SYSTEM SystemTests
  (* Version 1.0, 2018-08-29, Alois Zoitl, Johannes Kepler University, initial API and implementation and/or initial documentation *)
  APPLICATION Timing (* Small test application for measuring the execution time of a few fbs for evaluating runtime performance *)
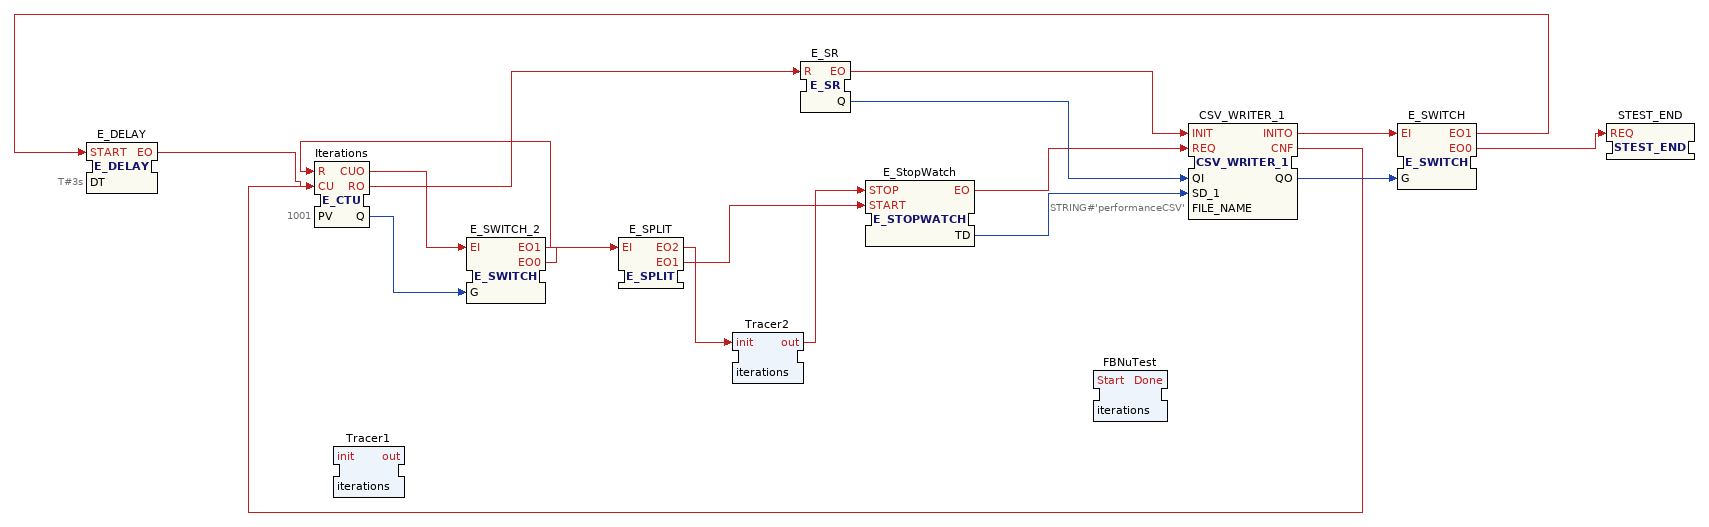
    FBS
      CSV_WRITER_1 : CSV_WRITER_1(FILE_NAME := STRING#'performanceCSV');
      E_SR : E_SR;
      E_SWITCH_2 : E_SWITCH;
      Iterations : E_CTU(PV := 1001);
      STEST_END : STEST_END;
      E_SWITCH : E_SWITCH;
      E_StopWatch : E_STOPWATCH;
      E_SPLIT : E_SPLIT;
      E_DELAY : E_DELAY(DT := T#3s);
    END_FBS
    SUBAPPLICATION FBNuTest
      EVENT_INPUT
        Start;
      END_EVENT
      EVENT_OUTPUT
        Done;
      END_EVENT
      VAR_INPUT
        iterations : UINT := UINT#100;
      END_VAR
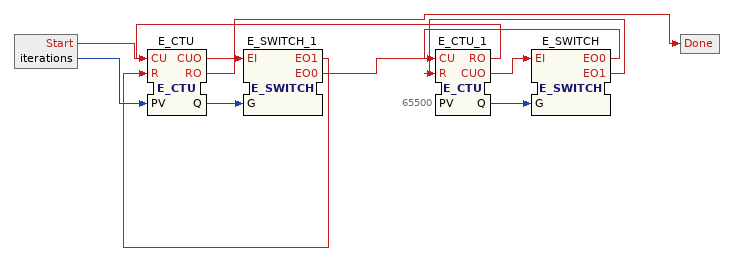
      FBS
        E_CTU : E_CTU;
        E_SWITCH_1 : E_SWITCH;
        E_SWITCH : E_SWITCH;
        E_CTU_1 : E_CTU(PV := 65500);
      END_FBS
      EVENT_CONNECTIONS
        E_CTU_1.RO TO E_CTU.CU;
        E_SWITCH_1.EO1 TO E_CTU.R;
        E_CTU.CUO TO E_SWITCH_1.EI;
        E_SWITCH_1.EO0 TO E_CTU_1.CU;
        E_CTU_1.CUO TO E_SWITCH.EI;
        E_SWITCH.EO0 TO E_CTU_1.CU;
        E_SWITCH.EO1 TO E_CTU_1.R;
        Start TO E_CTU.CU;
        E_CTU.RO TO Done;
      END_CONNECTIONS
      DATA_CONNECTIONS
        E_CTU.Q TO E_SWITCH_1.G;
        E_CTU_1.Q TO E_SWITCH.G;
        iterations TO E_CTU.PV;
      END_CONNECTIONS
    END_SUBAPPLICATION
    SUBAPPLICATION Tracer1
      EVENT_INPUT
        init;
      END_EVENT
      EVENT_OUTPUT
        out;
      END_EVENT
      VAR_INPUT
        iterations : UINT := UINT#1000;
      END_VAR
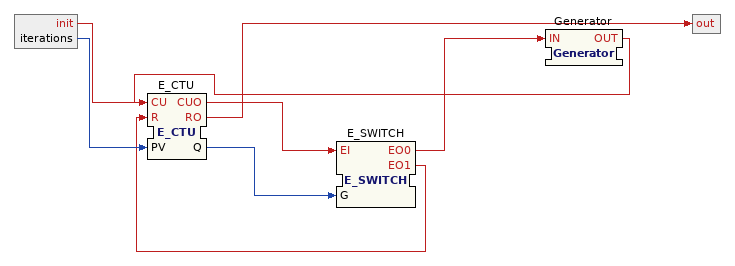
      FBS
        Generator : performance::Generator;
        E_CTU : E_CTU;
        E_SWITCH : E_SWITCH;
      END_FBS
      EVENT_CONNECTIONS
        init TO E_CTU.CU;
        E_CTU.CUO TO E_SWITCH.EI;
        E_SWITCH.EO0 TO Generator.IN;
        E_CTU.RO TO out;
        Generator.OUT TO E_CTU.CU;
        E_SWITCH.EO1 TO E_CTU.R;
      END_CONNECTIONS
      DATA_CONNECTIONS
        iterations TO E_CTU.PV;
        E_CTU.Q TO E_SWITCH.G;
      END_CONNECTIONS
    END_SUBAPPLICATION
    SUBAPPLICATION Tracer2
      EVENT_INPUT
        init;
      END_EVENT
      EVENT_OUTPUT
        out;
      END_EVENT
      VAR_INPUT
        iterations : UINT := UINT#1001;
      END_VAR
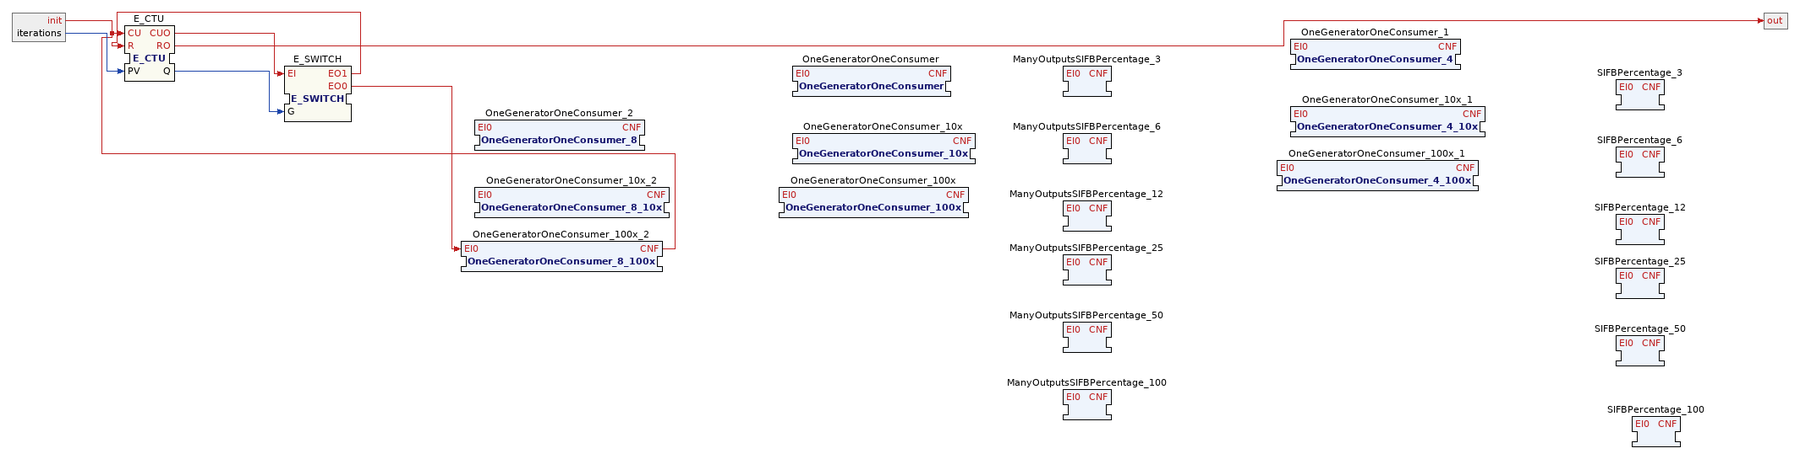
      FBS
        E_CTU : E_CTU;
        E_SWITCH : E_SWITCH;
      END_FBS
      SUBAPPS
        OneGeneratorOneConsumer : OneGeneratorOneConsumer;
        OneGeneratorOneConsumer_10x : OneGeneratorOneConsumer_10x;
        OneGeneratorOneConsumer_100x : OneGeneratorOneConsumer_100x;
        OneGeneratorOneConsumer_1 : OneGeneratorOneConsumer_4;
        OneGeneratorOneConsumer_10x_1 : OneGeneratorOneConsumer_4_10x;
        OneGeneratorOneConsumer_100x_1 : OneGeneratorOneConsumer_4_100x;
        OneGeneratorOneConsumer_100x_2 : OneGeneratorOneConsumer_8_100x;
        OneGeneratorOneConsumer_2 : OneGeneratorOneConsumer_8;
        OneGeneratorOneConsumer_10x_2 : OneGeneratorOneConsumer_8_10x;
      END_SUBAPPS
      SUBAPPLICATION SIFBPercentage_3
        {SET_ATTRIBUTE(Attribute1, )}
        EVENT_INPUT
          EI0;
        END_EVENT
        EVENT_OUTPUT
          CNF;
        END_EVENT
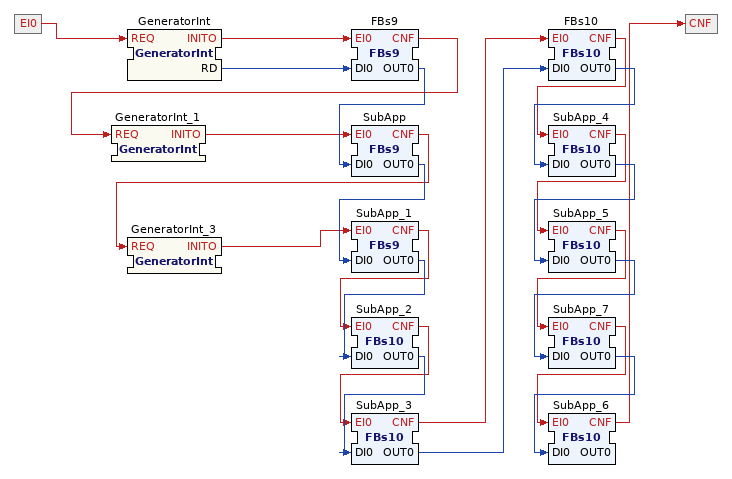
        FBS
          GeneratorInt : performance::GeneratorInt;
          GeneratorInt_1 : performance::GeneratorInt;
          GeneratorInt_3 : performance::GeneratorInt;
        END_FBS
        SUBAPPS
          FBs9 : FBs9;
          SubApp : FBs9;
          SubApp_1 : FBs9;
          SubApp_2 : FBs10;
          SubApp_3 : FBs10;
          SubApp_4 : FBs10;
          SubApp_5 : FBs10;
          SubApp_6 : FBs10;
          SubApp_7 : FBs10;
          FBs10 : FBs10;
        END_SUBAPPS
        EVENT_CONNECTIONS
          EI0 TO GeneratorInt.REQ;
          SubApp_2.CNF TO SubApp_3.EI0;
          SubApp_4.CNF TO SubApp_5.EI0;
          SubApp_5.CNF TO SubApp_7.EI0;
          SubApp_7.CNF TO SubApp_6.EI0;
          SubApp_3.CNF TO FBs10.EI0;
          FBs10.CNF TO SubApp_4.EI0;
          SubApp_6.CNF TO CNF;
          FBs9.CNF TO GeneratorInt_1.REQ;
          SubApp.CNF TO GeneratorInt_3.REQ;
          GeneratorInt_1.INITO TO SubApp.EI0;
          GeneratorInt.INITO TO FBs9.EI0;
          GeneratorInt_3.INITO TO SubApp_1.EI0;
          SubApp_1.CNF TO SubApp_2.EI0;
        END_CONNECTIONS
        DATA_CONNECTIONS
          SubApp_2.OUT0 TO SubApp_3.DI0;
          SubApp_1.OUT0 TO SubApp_2.DI0;
          SubApp.OUT0 TO SubApp_1.DI0;
          SubApp_7.OUT0 TO SubApp_6.DI0;
          SubApp_4.OUT0 TO SubApp_5.DI0;
          SubApp_5.OUT0 TO SubApp_7.DI0;
          FBs10.OUT0 TO SubApp_4.DI0;
          SubApp_3.OUT0 TO FBs10.DI0;
          GeneratorInt.RD TO FBs9.DI0;
          FBs9.OUT0 TO SubApp.DI0;
        END_CONNECTIONS
      END_SUBAPPLICATION
      SUBAPPLICATION SIFBPercentage_6
        {SET_ATTRIBUTE(Attribute1, )}
        EVENT_INPUT
          EI0;
        END_EVENT
        EVENT_OUTPUT
          CNF;
        END_EVENT
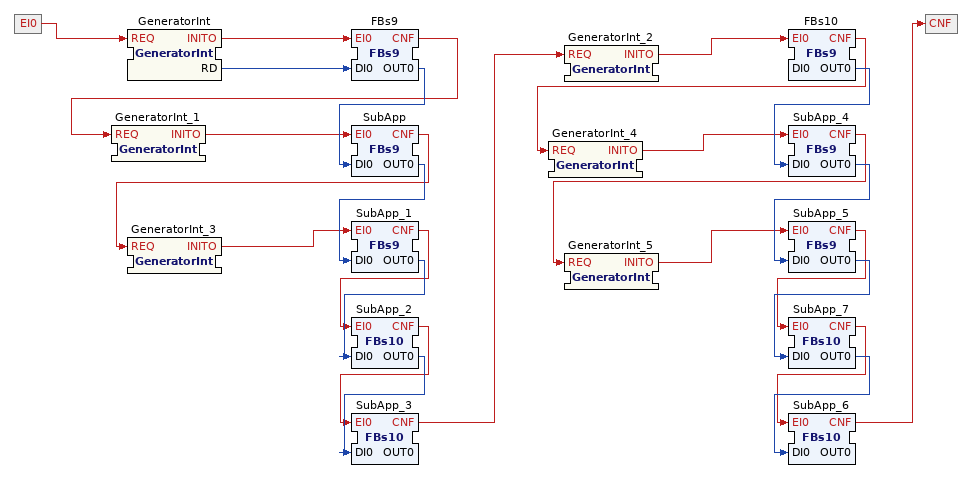
        FBS
          GeneratorInt : performance::GeneratorInt;
          GeneratorInt_1 : performance::GeneratorInt;
          GeneratorInt_3 : performance::GeneratorInt;
          GeneratorInt_2 : performance::GeneratorInt;
          GeneratorInt_4 : performance::GeneratorInt;
          GeneratorInt_5 : performance::GeneratorInt;
        END_FBS
        SUBAPPS
          FBs9 : FBs9;
          SubApp : FBs9;
          SubApp_1 : FBs9;
          SubApp_2 : FBs10;
          SubApp_3 : FBs10;
          SubApp_4 : FBs9;
          SubApp_5 : FBs9;
          SubApp_6 : FBs10;
          SubApp_7 : FBs10;
          FBs10 : FBs9;
        END_SUBAPPS
        EVENT_CONNECTIONS
          EI0 TO GeneratorInt.REQ;
          SubApp_2.CNF TO SubApp_3.EI0;
          SubApp_4.CNF TO GeneratorInt_5.REQ;
          SubApp_5.CNF TO SubApp_7.EI0;
          SubApp_7.CNF TO SubApp_6.EI0;
          FBs10.CNF TO GeneratorInt_4.REQ;
          SubApp_6.CNF TO CNF;
          FBs9.CNF TO GeneratorInt_1.REQ;
          SubApp.CNF TO GeneratorInt_3.REQ;
          GeneratorInt_1.INITO TO SubApp.EI0;
          GeneratorInt.INITO TO FBs9.EI0;
          GeneratorInt_3.INITO TO SubApp_1.EI0;
          GeneratorInt_2.INITO TO FBs10.EI0;
          GeneratorInt_4.INITO TO SubApp_4.EI0;
          GeneratorInt_5.INITO TO SubApp_5.EI0;
          SubApp_3.CNF TO GeneratorInt_2.REQ;
          SubApp_1.CNF TO SubApp_2.EI0;
        END_CONNECTIONS
        DATA_CONNECTIONS
          SubApp_2.OUT0 TO SubApp_3.DI0;
          SubApp_1.OUT0 TO SubApp_2.DI0;
          SubApp.OUT0 TO SubApp_1.DI0;
          SubApp_7.OUT0 TO SubApp_6.DI0;
          SubApp_4.OUT0 TO SubApp_5.DI0;
          SubApp_5.OUT0 TO SubApp_7.DI0;
          FBs10.OUT0 TO SubApp_4.DI0;
          GeneratorInt.RD TO FBs9.DI0;
          FBs9.OUT0 TO SubApp.DI0;
        END_CONNECTIONS
      END_SUBAPPLICATION
      SUBAPPLICATION SIFBPercentage_12
        {SET_ATTRIBUTE(Attribute1, )}
        EVENT_INPUT
          EI0;
        END_EVENT
        EVENT_OUTPUT
          CNF;
        END_EVENT
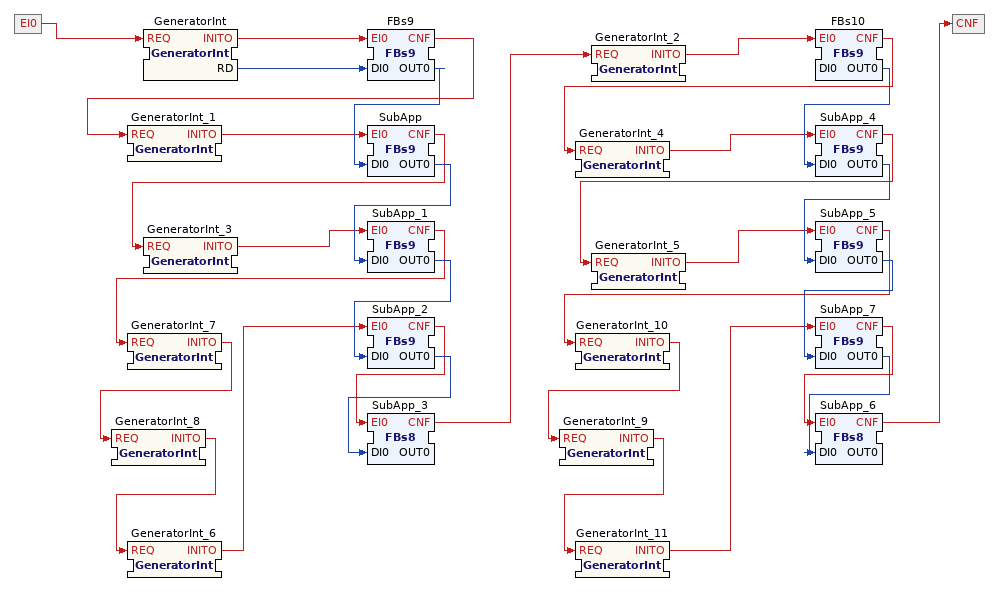
        FBS
          GeneratorInt : performance::GeneratorInt;
          GeneratorInt_1 : performance::GeneratorInt;
          GeneratorInt_3 : performance::GeneratorInt;
          GeneratorInt_2 : performance::GeneratorInt;
          GeneratorInt_4 : performance::GeneratorInt;
          GeneratorInt_5 : performance::GeneratorInt;
          GeneratorInt_6 : performance::GeneratorInt;
          GeneratorInt_7 : performance::GeneratorInt;
          GeneratorInt_8 : performance::GeneratorInt;
          GeneratorInt_9 : performance::GeneratorInt;
          GeneratorInt_10 : performance::GeneratorInt;
          GeneratorInt_11 : performance::GeneratorInt;
        END_FBS
        SUBAPPS
          FBs9 : FBs9;
          SubApp : FBs9;
          SubApp_1 : FBs9;
          SubApp_2 : FBs9;
          SubApp_3 : FBs8;
          SubApp_4 : FBs9;
          SubApp_5 : FBs9;
          SubApp_6 : FBs8;
          SubApp_7 : FBs9;
          FBs10 : FBs9;
        END_SUBAPPS
        EVENT_CONNECTIONS
          EI0 TO GeneratorInt.REQ;
          SubApp_2.CNF TO SubApp_3.EI0;
          SubApp_4.CNF TO GeneratorInt_5.REQ;
          SubApp_5.CNF TO GeneratorInt_10.REQ;
          SubApp_7.CNF TO SubApp_6.EI0;
          FBs10.CNF TO GeneratorInt_4.REQ;
          SubApp_6.CNF TO CNF;
          FBs9.CNF TO GeneratorInt_1.REQ;
          SubApp.CNF TO GeneratorInt_3.REQ;
          GeneratorInt_1.INITO TO SubApp.EI0;
          GeneratorInt.INITO TO FBs9.EI0;
          GeneratorInt_3.INITO TO SubApp_1.EI0;
          GeneratorInt_2.INITO TO FBs10.EI0;
          GeneratorInt_4.INITO TO SubApp_4.EI0;
          GeneratorInt_5.INITO TO SubApp_5.EI0;
          SubApp_3.CNF TO GeneratorInt_2.REQ;
          SubApp_1.CNF TO GeneratorInt_7.REQ;
          GeneratorInt_7.INITO TO GeneratorInt_8.REQ;
          GeneratorInt_8.INITO TO GeneratorInt_6.REQ;
          GeneratorInt_6.INITO TO SubApp_2.EI0;
          GeneratorInt_10.INITO TO GeneratorInt_9.REQ;
          GeneratorInt_9.INITO TO GeneratorInt_11.REQ;
          GeneratorInt_11.INITO TO SubApp_7.EI0;
        END_CONNECTIONS
        DATA_CONNECTIONS
          SubApp_2.OUT0 TO SubApp_3.DI0;
          SubApp_1.OUT0 TO SubApp_2.DI0;
          SubApp.OUT0 TO SubApp_1.DI0;
          SubApp_7.OUT0 TO SubApp_6.DI0;
          SubApp_4.OUT0 TO SubApp_5.DI0;
          SubApp_5.OUT0 TO SubApp_7.DI0;
          FBs10.OUT0 TO SubApp_4.DI0;
          GeneratorInt.RD TO FBs9.DI0;
          FBs9.OUT0 TO SubApp.DI0;
        END_CONNECTIONS
      END_SUBAPPLICATION
      SUBAPPLICATION SIFBPercentage_25
        {SET_ATTRIBUTE(Attribute1, )}
        EVENT_INPUT
          EI0;
        END_EVENT
        EVENT_OUTPUT
          CNF;
        END_EVENT
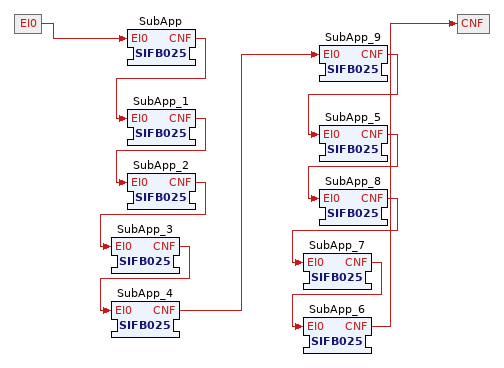
        SUBAPPS
          SubApp : SIFB025;
          SubApp_1 : SIFB025;
          SubApp_2 : SIFB025;
          SubApp_3 : SIFB025;
          SubApp_4 : SIFB025;
          SubApp_5 : SIFB025;
          SubApp_6 : SIFB025;
          SubApp_7 : SIFB025;
          SubApp_8 : SIFB025;
          SubApp_9 : SIFB025;
        END_SUBAPPS
        EVENT_CONNECTIONS
          SubApp_3.CNF TO SubApp_4.EI0;
          SubApp_2.CNF TO SubApp_3.EI0;
          SubApp_1.CNF TO SubApp_2.EI0;
          SubApp.CNF TO SubApp_1.EI0;
          SubApp_5.CNF TO SubApp_8.EI0;
          SubApp_8.CNF TO SubApp_7.EI0;
          SubApp_7.CNF TO SubApp_6.EI0;
          SubApp_9.CNF TO SubApp_5.EI0;
          SubApp_4.CNF TO SubApp_9.EI0;
          EI0 TO SubApp.EI0;
          SubApp_6.CNF TO CNF;
        END_CONNECTIONS
      END_SUBAPPLICATION
      SUBAPPLICATION SIFBPercentage_50
        {SET_ATTRIBUTE(Attribute1, )}
        EVENT_INPUT
          EI0;
        END_EVENT
        EVENT_OUTPUT
          CNF;
        END_EVENT
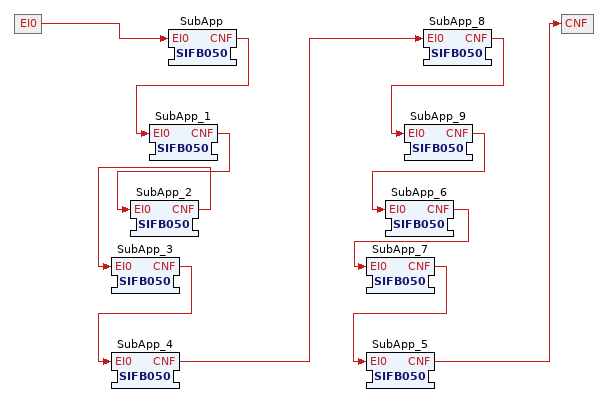
        SUBAPPS
          SubApp : SIFB050;
          SubApp_1 : SIFB050;
          SubApp_2 : SIFB050;
          SubApp_3 : SIFB050;
          SubApp_4 : SIFB050;
          SubApp_5 : SIFB050;
          SubApp_6 : SIFB050;
          SubApp_7 : SIFB050;
          SubApp_8 : SIFB050;
          SubApp_9 : SIFB050;
        END_SUBAPPS
        EVENT_CONNECTIONS
          SubApp.CNF TO SubApp_1.EI0;
          SubApp_1.CNF TO SubApp_2.EI0;
          SubApp_2.CNF TO SubApp_3.EI0;
          SubApp_3.CNF TO SubApp_4.EI0;
          SubApp_8.CNF TO SubApp_9.EI0;
          SubApp_9.CNF TO SubApp_6.EI0;
          SubApp_7.CNF TO SubApp_5.EI0;
          SubApp_6.CNF TO SubApp_7.EI0;
          SubApp_5.CNF TO CNF;
          EI0 TO SubApp.EI0;
          SubApp_4.CNF TO SubApp_8.EI0;
        END_CONNECTIONS
      END_SUBAPPLICATION
      SUBAPPLICATION SIFBPercentage_100
        {SET_ATTRIBUTE(Attribute1, )}
        EVENT_INPUT
          EI0;
        END_EVENT
        EVENT_OUTPUT
          CNF;
        END_EVENT
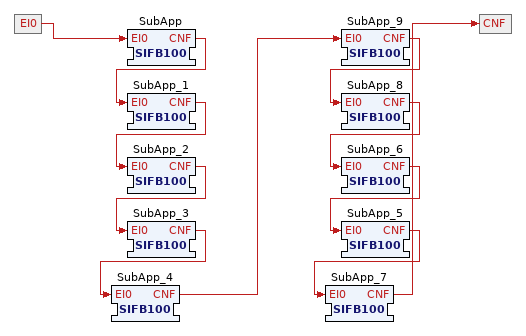
        SUBAPPS
          SubApp : SIFB100;
          SubApp_1 : SIFB100;
          SubApp_2 : SIFB100;
          SubApp_3 : SIFB100;
          SubApp_4 : SIFB100;
          SubApp_5 : SIFB100;
          SubApp_6 : SIFB100;
          SubApp_7 : SIFB100;
          SubApp_8 : SIFB100;
          SubApp_9 : SIFB100;
        END_SUBAPPS
        EVENT_CONNECTIONS
          SubApp.CNF TO SubApp_1.EI0;
          SubApp_1.CNF TO SubApp_2.EI0;
          SubApp_2.CNF TO SubApp_3.EI0;
          SubApp_3.CNF TO SubApp_4.EI0;
          SubApp_8.CNF TO SubApp_6.EI0;
          SubApp_6.CNF TO SubApp_5.EI0;
          SubApp_5.CNF TO SubApp_7.EI0;
          SubApp_9.CNF TO SubApp_8.EI0;
          SubApp_4.CNF TO SubApp_9.EI0;
          EI0 TO SubApp.EI0;
          SubApp_7.CNF TO CNF;
        END_CONNECTIONS
      END_SUBAPPLICATION
      SUBAPPLICATION ManyOutputsSIFBPercentage_12
        {SET_ATTRIBUTE(Attribute1, )}
        EVENT_INPUT
          EI0;
        END_EVENT
        EVENT_OUTPUT
          CNF;
        END_EVENT
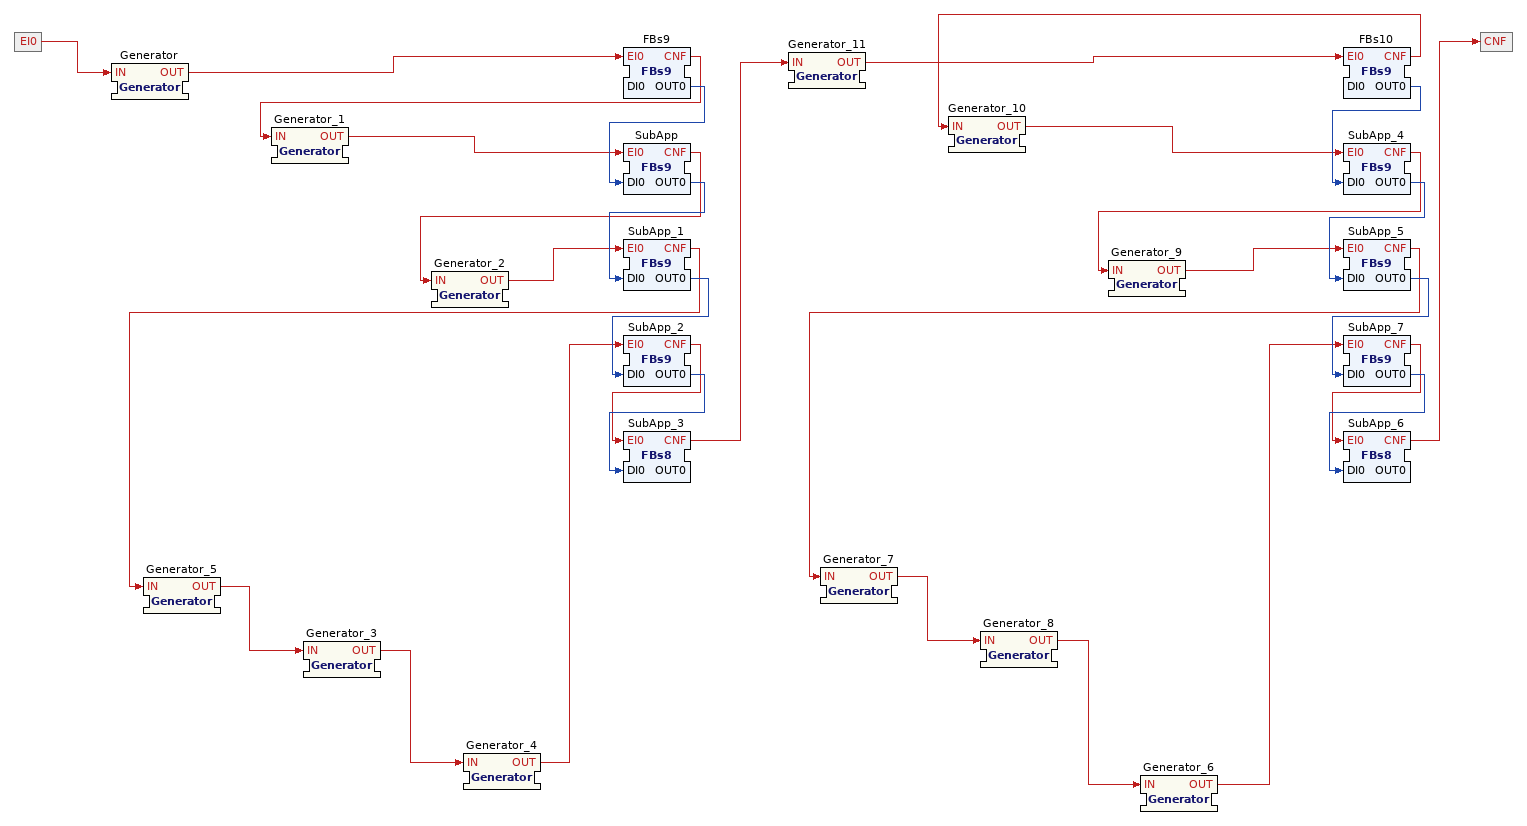
        FBS
          Generator : performance::Generator;
          Generator_1 : performance::Generator;
          Generator_2 : performance::Generator;
          Generator_3 : performance::Generator;
          Generator_4 : performance::Generator;
          Generator_5 : performance::Generator;
          Generator_6 : performance::Generator;
          Generator_7 : performance::Generator;
          Generator_8 : performance::Generator;
          Generator_9 : performance::Generator;
          Generator_10 : performance::Generator;
          Generator_11 : performance::Generator;
        END_FBS
        SUBAPPS
          FBs9 : FBs9;
          SubApp : FBs9;
          SubApp_1 : FBs9;
          SubApp_2 : FBs9;
          SubApp_3 : FBs8;
          SubApp_4 : FBs9;
          SubApp_5 : FBs9;
          SubApp_6 : FBs8;
          SubApp_7 : FBs9;
          FBs10 : FBs9;
        END_SUBAPPS
        EVENT_CONNECTIONS
          SubApp_2.CNF TO SubApp_3.EI0;
          SubApp_7.CNF TO SubApp_6.EI0;
          SubApp_6.CNF TO CNF;
          EI0 TO Generator.IN;
          Generator.OUT TO FBs9.EI0;
          FBs9.CNF TO Generator_1.IN;
          SubApp.CNF TO Generator_2.IN;
          Generator_2.OUT TO SubApp_1.EI0;
          SubApp_1.CNF TO Generator_5.IN;
          Generator_5.OUT TO Generator_3.IN;
          Generator_3.OUT TO Generator_4.IN;
          Generator_4.OUT TO SubApp_2.EI0;
          SubApp_3.CNF TO Generator_11.IN;
          Generator_11.OUT TO FBs10.EI0;
          FBs10.CNF TO Generator_10.IN;
          Generator_10.OUT TO SubApp_4.EI0;
          SubApp_4.CNF TO Generator_9.IN;
          Generator_9.OUT TO SubApp_5.EI0;
          SubApp_5.CNF TO Generator_7.IN;
          Generator_7.OUT TO Generator_8.IN;
          Generator_8.OUT TO Generator_6.IN;
          Generator_6.OUT TO SubApp_7.EI0;
          Generator_1.OUT TO SubApp.EI0;
        END_CONNECTIONS
        DATA_CONNECTIONS
          SubApp_2.OUT0 TO SubApp_3.DI0;
          SubApp_1.OUT0 TO SubApp_2.DI0;
          SubApp.OUT0 TO SubApp_1.DI0;
          SubApp_7.OUT0 TO SubApp_6.DI0;
          SubApp_4.OUT0 TO SubApp_5.DI0;
          SubApp_5.OUT0 TO SubApp_7.DI0;
          FBs10.OUT0 TO SubApp_4.DI0;
          FBs9.OUT0 TO SubApp.DI0;
        END_CONNECTIONS
      END_SUBAPPLICATION
      SUBAPPLICATION ManyOutputsSIFBPercentage_100
        {SET_ATTRIBUTE(Attribute1, )}
        EVENT_INPUT
          EI0;
        END_EVENT
        EVENT_OUTPUT
          CNF;
        END_EVENT
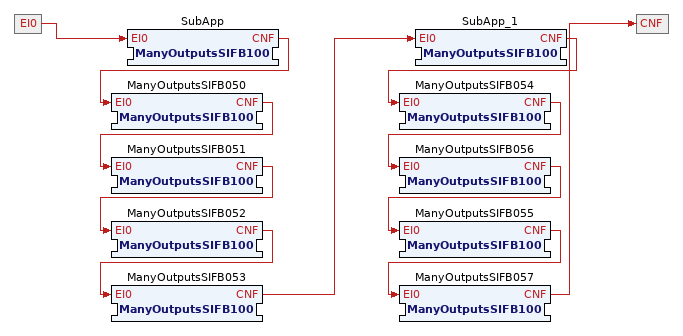
        SUBAPPS
          SubApp : ManyOutputsSIFB100;
          ManyOutputsSIFB050 : ManyOutputsSIFB100;
          ManyOutputsSIFB051 : ManyOutputsSIFB100;
          ManyOutputsSIFB052 : ManyOutputsSIFB100;
          ManyOutputsSIFB053 : ManyOutputsSIFB100;
          ManyOutputsSIFB054 : ManyOutputsSIFB100;
          ManyOutputsSIFB055 : ManyOutputsSIFB100;
          ManyOutputsSIFB056 : ManyOutputsSIFB100;
          ManyOutputsSIFB057 : ManyOutputsSIFB100;
          SubApp_1 : ManyOutputsSIFB100;
        END_SUBAPPS
        EVENT_CONNECTIONS
          EI0 TO SubApp.EI0;
          SubApp.CNF TO ManyOutputsSIFB050.EI0;
          ManyOutputsSIFB050.CNF TO ManyOutputsSIFB051.EI0;
          ManyOutputsSIFB051.CNF TO ManyOutputsSIFB052.EI0;
          ManyOutputsSIFB052.CNF TO ManyOutputsSIFB053.EI0;
          ManyOutputsSIFB056.CNF TO ManyOutputsSIFB055.EI0;
          ManyOutputsSIFB054.CNF TO ManyOutputsSIFB056.EI0;
          SubApp_1.CNF TO ManyOutputsSIFB054.EI0;
          ManyOutputsSIFB055.CNF TO ManyOutputsSIFB057.EI0;
          ManyOutputsSIFB053.CNF TO SubApp_1.EI0;
          ManyOutputsSIFB057.CNF TO CNF;
        END_CONNECTIONS
      END_SUBAPPLICATION
      SUBAPPLICATION ManyOutputsSIFBPercentage_6
        {SET_ATTRIBUTE(Attribute1, )}
        EVENT_INPUT
          EI0;
        END_EVENT
        EVENT_OUTPUT
          CNF;
        END_EVENT
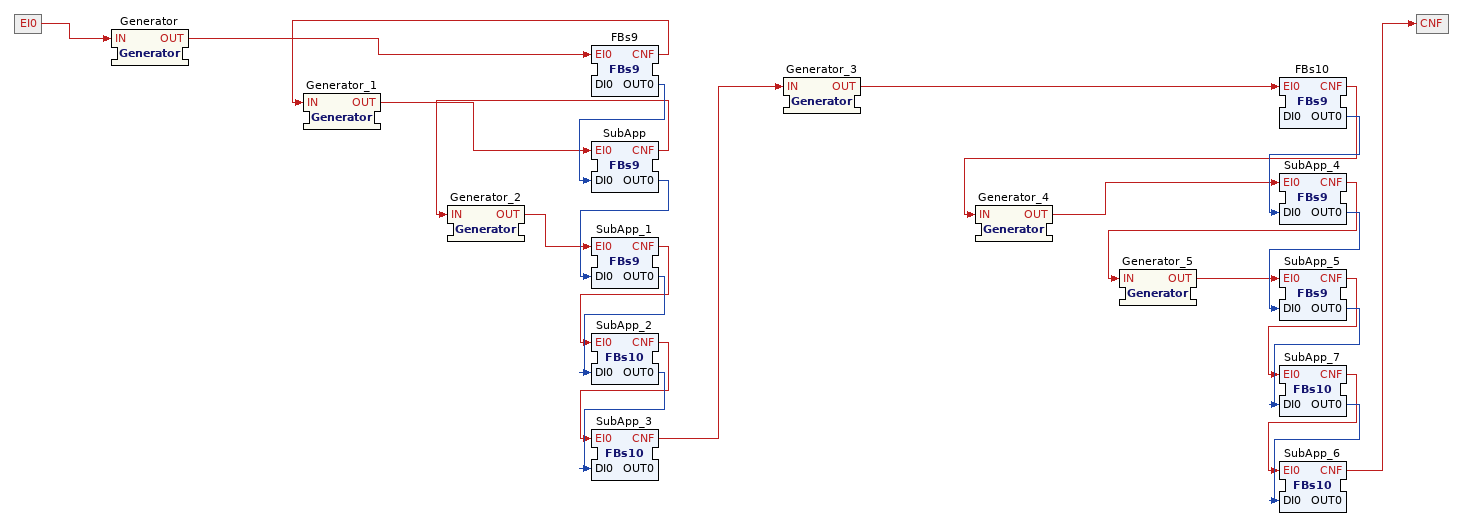
        FBS
          Generator : performance::Generator;
          Generator_1 : performance::Generator;
          Generator_2 : performance::Generator;
          Generator_3 : performance::Generator;
          Generator_4 : performance::Generator;
          Generator_5 : performance::Generator;
        END_FBS
        SUBAPPS
          FBs9 : FBs9;
          SubApp : FBs9;
          SubApp_1 : FBs9;
          SubApp_2 : FBs10;
          SubApp_3 : FBs10;
          SubApp_4 : FBs9;
          SubApp_5 : FBs9;
          SubApp_6 : FBs10;
          SubApp_7 : FBs10;
          FBs10 : FBs9;
        END_SUBAPPS
        EVENT_CONNECTIONS
          SubApp_2.CNF TO SubApp_3.EI0;
          SubApp_5.CNF TO SubApp_7.EI0;
          SubApp_7.CNF TO SubApp_6.EI0;
          SubApp_6.CNF TO CNF;
          SubApp_1.CNF TO SubApp_2.EI0;
          Generator.OUT TO FBs9.EI0;
          FBs9.CNF TO Generator_1.IN;
          Generator_2.OUT TO SubApp_1.EI0;
          Generator_1.OUT TO SubApp.EI0;
          EI0 TO Generator.IN;
          SubApp_3.CNF TO Generator_3.IN;
          Generator_3.OUT TO FBs10.EI0;
          Generator_4.OUT TO SubApp_4.EI0;
          FBs10.CNF TO Generator_4.IN;
          Generator_5.OUT TO SubApp_5.EI0;
          SubApp_4.CNF TO Generator_5.IN;
          SubApp.CNF TO Generator_2.IN;
        END_CONNECTIONS
        DATA_CONNECTIONS
          SubApp_2.OUT0 TO SubApp_3.DI0;
          SubApp_1.OUT0 TO SubApp_2.DI0;
          SubApp.OUT0 TO SubApp_1.DI0;
          SubApp_7.OUT0 TO SubApp_6.DI0;
          SubApp_4.OUT0 TO SubApp_5.DI0;
          SubApp_5.OUT0 TO SubApp_7.DI0;
          FBs10.OUT0 TO SubApp_4.DI0;
          FBs9.OUT0 TO SubApp.DI0;
        END_CONNECTIONS
      END_SUBAPPLICATION
      SUBAPPLICATION ManyOutputsSIFBPercentage_3
        {SET_ATTRIBUTE(Attribute1, )}
        EVENT_INPUT
          EI0;
        END_EVENT
        EVENT_OUTPUT
          CNF;
        END_EVENT
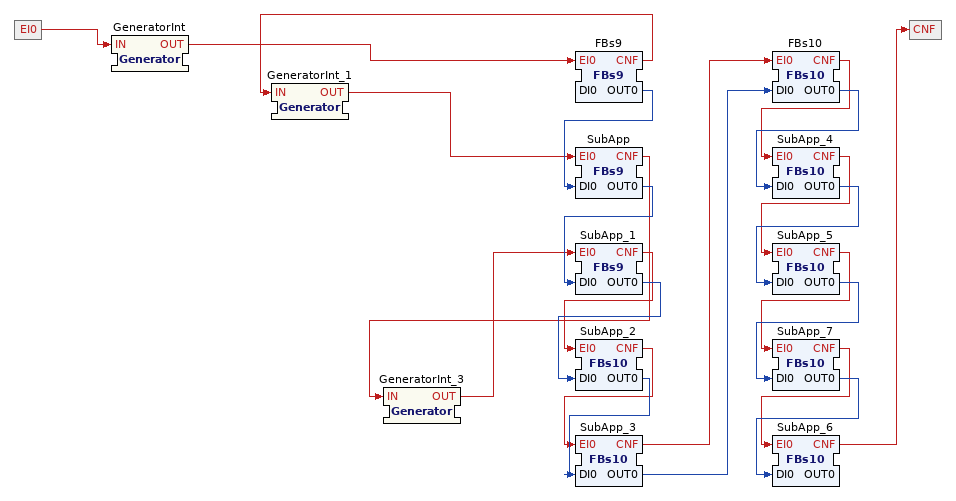
        FBS
          GeneratorInt : performance::Generator;
          GeneratorInt_1 : performance::Generator;
          GeneratorInt_3 : performance::Generator;
        END_FBS
        SUBAPPS
          FBs9 : FBs9;
          SubApp : FBs9;
          SubApp_1 : FBs9;
          SubApp_2 : FBs10;
          SubApp_3 : FBs10;
          SubApp_4 : FBs10;
          SubApp_5 : FBs10;
          SubApp_6 : FBs10;
          SubApp_7 : FBs10;
          FBs10 : FBs10;
        END_SUBAPPS
        EVENT_CONNECTIONS
          SubApp_2.CNF TO SubApp_3.EI0;
          SubApp_4.CNF TO SubApp_5.EI0;
          SubApp_5.CNF TO SubApp_7.EI0;
          SubApp_7.CNF TO SubApp_6.EI0;
          SubApp_3.CNF TO FBs10.EI0;
          FBs10.CNF TO SubApp_4.EI0;
          SubApp_6.CNF TO CNF;
          SubApp_1.CNF TO SubApp_2.EI0;
          GeneratorInt.OUT TO FBs9.EI0;
          FBs9.CNF TO GeneratorInt_1.IN;
          GeneratorInt_1.OUT TO SubApp.EI0;
          SubApp.CNF TO GeneratorInt_3.IN;
          GeneratorInt_3.OUT TO SubApp_1.EI0;
          EI0 TO GeneratorInt.IN;
        END_CONNECTIONS
        DATA_CONNECTIONS
          SubApp_2.OUT0 TO SubApp_3.DI0;
          SubApp_1.OUT0 TO SubApp_2.DI0;
          SubApp.OUT0 TO SubApp_1.DI0;
          SubApp_7.OUT0 TO SubApp_6.DI0;
          SubApp_4.OUT0 TO SubApp_5.DI0;
          SubApp_5.OUT0 TO SubApp_7.DI0;
          FBs10.OUT0 TO SubApp_4.DI0;
          SubApp_3.OUT0 TO FBs10.DI0;
          FBs9.OUT0 TO SubApp.DI0;
        END_CONNECTIONS
      END_SUBAPPLICATION
      SUBAPPLICATION ManyOutputsSIFBPercentage_50
        {SET_ATTRIBUTE(Attribute1, )}
        EVENT_INPUT
          EI0;
        END_EVENT
        EVENT_OUTPUT
          CNF;
        END_EVENT
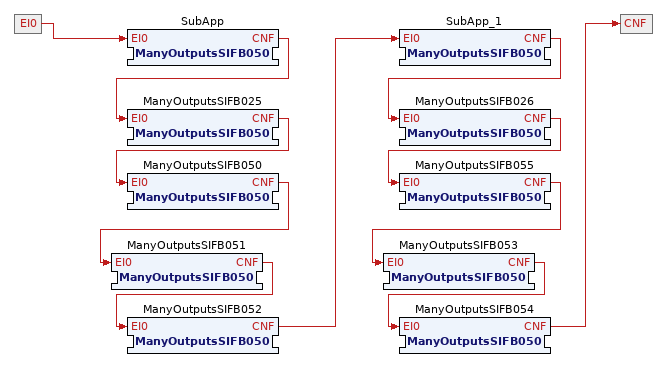
        SUBAPPS
          SubApp : ManyOutputsSIFB050;
          ManyOutputsSIFB025 : ManyOutputsSIFB050;
          ManyOutputsSIFB050 : ManyOutputsSIFB050;
          ManyOutputsSIFB051 : ManyOutputsSIFB050;
          ManyOutputsSIFB052 : ManyOutputsSIFB050;
          ManyOutputsSIFB053 : ManyOutputsSIFB050;
          ManyOutputsSIFB026 : ManyOutputsSIFB050;
          SubApp_1 : ManyOutputsSIFB050;
          ManyOutputsSIFB054 : ManyOutputsSIFB050;
          ManyOutputsSIFB055 : ManyOutputsSIFB050;
        END_SUBAPPS
        EVENT_CONNECTIONS
          SubApp.CNF TO ManyOutputsSIFB025.EI0;
          ManyOutputsSIFB025.CNF TO ManyOutputsSIFB050.EI0;
          ManyOutputsSIFB050.CNF TO ManyOutputsSIFB051.EI0;
          ManyOutputsSIFB051.CNF TO ManyOutputsSIFB052.EI0;
          ManyOutputsSIFB053.CNF TO ManyOutputsSIFB054.EI0;
          SubApp_1.CNF TO ManyOutputsSIFB026.EI0;
          ManyOutputsSIFB055.CNF TO ManyOutputsSIFB053.EI0;
          ManyOutputsSIFB026.CNF TO ManyOutputsSIFB055.EI0;
          ManyOutputsSIFB052.CNF TO SubApp_1.EI0;
          EI0 TO SubApp.EI0;
          ManyOutputsSIFB054.CNF TO CNF;
        END_CONNECTIONS
      END_SUBAPPLICATION
      SUBAPPLICATION ManyOutputsSIFBPercentage_25
        {SET_ATTRIBUTE(Attribute1, )}
        EVENT_INPUT
          EI0;
        END_EVENT
        EVENT_OUTPUT
          CNF;
        END_EVENT
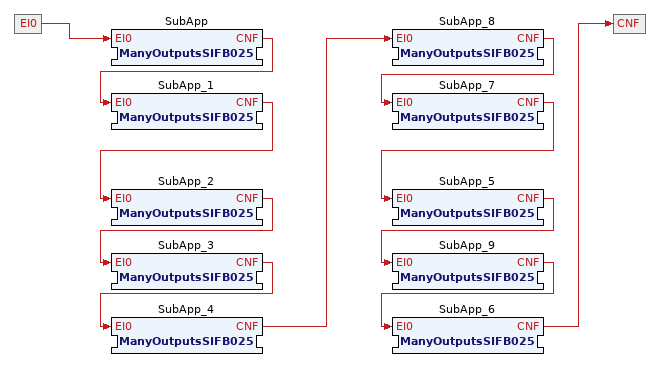
        SUBAPPS
          SubApp : ManyOutputsSIFB025;
          SubApp_1 : ManyOutputsSIFB025;
          SubApp_2 : ManyOutputsSIFB025;
          SubApp_3 : ManyOutputsSIFB025;
          SubApp_4 : ManyOutputsSIFB025;
          SubApp_5 : ManyOutputsSIFB025;
          SubApp_6 : ManyOutputsSIFB025;
          SubApp_7 : ManyOutputsSIFB025;
          SubApp_8 : ManyOutputsSIFB025;
          SubApp_9 : ManyOutputsSIFB025;
        END_SUBAPPS
        EVENT_CONNECTIONS
          SubApp.CNF TO SubApp_1.EI0;
          SubApp_1.CNF TO SubApp_2.EI0;
          SubApp_2.CNF TO SubApp_3.EI0;
          SubApp_3.CNF TO SubApp_4.EI0;
          SubApp_8.CNF TO SubApp_7.EI0;
          SubApp_7.CNF TO SubApp_5.EI0;
          SubApp_9.CNF TO SubApp_6.EI0;
          SubApp_5.CNF TO SubApp_9.EI0;
          SubApp_4.CNF TO SubApp_8.EI0;
          EI0 TO SubApp.EI0;
          SubApp_6.CNF TO CNF;
        END_CONNECTIONS
      END_SUBAPPLICATION
      EVENT_CONNECTIONS
        init TO E_CTU.CU;
        E_CTU.CUO TO E_SWITCH.EI;
        E_CTU.RO TO out;
        E_SWITCH.EO1 TO E_CTU.R;
        E_SWITCH.EO0 TO OneGeneratorOneConsumer_100x_2.EI0;
        OneGeneratorOneConsumer_100x_2.CNF TO E_CTU.CU;
      END_CONNECTIONS
      DATA_CONNECTIONS
        iterations TO E_CTU.PV;
        E_CTU.Q TO E_SWITCH.G;
      END_CONNECTIONS
    END_SUBAPPLICATION
    EVENT_CONNECTIONS
      E_SR.EO TO CSV_WRITER_1.INIT;
      Iterations.CUO TO E_SWITCH_2.EI;
      E_SWITCH_2.EO1 TO Iterations.R;
      Iterations.RO TO E_SR.R;
      E_SWITCH.EO1 TO E_DELAY.START;
      E_SWITCH.EO0 TO STEST_END.REQ;
      CSV_WRITER_1.INITO TO E_SWITCH.EI;
      E_SWITCH_2.EO0 TO E_SPLIT.EI;
      E_StopWatch.EO TO CSV_WRITER_1.REQ;
      CSV_WRITER_1.CNF TO Iterations.CU;
      Tracer2.out TO E_StopWatch.STOP;
      E_SPLIT.EO2 TO Tracer2.init;
      E_SPLIT.EO1 TO E_StopWatch.START;
      E_DELAY.EO TO Iterations.CU;
    END_CONNECTIONS
    DATA_CONNECTIONS
      E_SR.Q TO CSV_WRITER_1.QI;
      Iterations.Q TO E_SWITCH_2.G;
      CSV_WRITER_1.QO TO E_SWITCH.G;
      E_StopWatch.TD TO CSV_WRITER_1.SD_1;
    END_CONNECTIONS
  END_APPLICATION
  APPLICATION Soft_Pass_Example
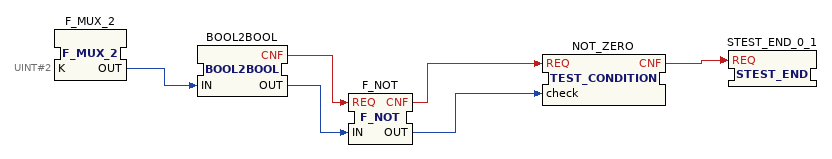
    FBS
      NOT_ZERO : TEST_CONDITION;
      STEST_END_0_1 : STEST_END;
      F_MUX_2 : F_MUX_2(K := UINT#2);
      F_NOT : F_NOT;
      BOOL2BOOL : BOOL2BOOL;
    END_FBS
    EVENT_CONNECTIONS
      F_NOT.CNF TO NOT_ZERO.REQ;
      NOT_ZERO.CNF TO STEST_END_0_1.REQ;
      BOOL2BOOL.CNF TO F_NOT.REQ;
    END_CONNECTIONS
    DATA_CONNECTIONS
      F_MUX_2.OUT TO BOOL2BOOL.IN;
      F_NOT.OUT TO NOT_ZERO.check;
      BOOL2BOOL.OUT TO F_NOT.IN;
    END_CONNECTIONS
  END_APPLICATION
  APPLICATION Fail_Example
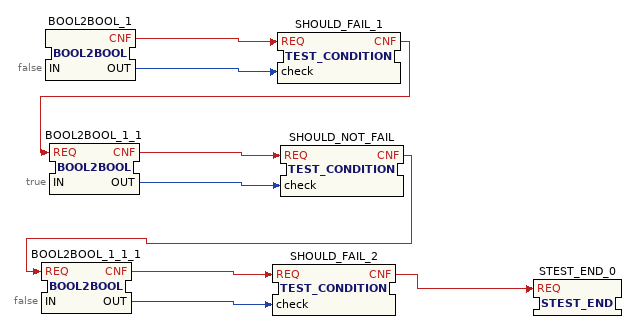
    FBS
      STEST_END_0 : STEST_END;
      BOOL2BOOL_1_1_1 : BOOL2BOOL(IN := false);
      SHOULD_FAIL_1 : TEST_CONDITION;
      BOOL2BOOL_1 : BOOL2BOOL(IN := false);
      SHOULD_NOT_FAIL : TEST_CONDITION;
      BOOL2BOOL_1_1 : BOOL2BOOL(IN := true);
      SHOULD_FAIL_2 : TEST_CONDITION;
    END_FBS
    EVENT_CONNECTIONS
      BOOL2BOOL_1.CNF TO SHOULD_FAIL_1.REQ;
      SHOULD_FAIL_2.CNF TO STEST_END_0.REQ;
      SHOULD_FAIL_1.CNF TO BOOL2BOOL_1_1.REQ;
      SHOULD_NOT_FAIL.CNF TO BOOL2BOOL_1_1_1.REQ;
      BOOL2BOOL_1_1_1.CNF TO SHOULD_FAIL_2.REQ;
      BOOL2BOOL_1_1.CNF TO SHOULD_NOT_FAIL.REQ;
    END_CONNECTIONS
    DATA_CONNECTIONS
      BOOL2BOOL_1_1.OUT TO SHOULD_NOT_FAIL.check;
      BOOL2BOOL_1.OUT TO SHOULD_FAIL_1.check;
      BOOL2BOOL_1_1_1.OUT TO SHOULD_FAIL_2.check;
    END_CONNECTIONS
  END_APPLICATION
  APPLICATION Hard_Pass_Example
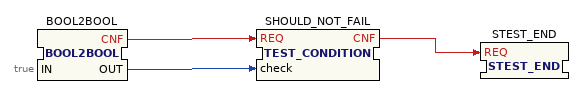
    FBS
      STEST_END : STEST_END;
      BOOL2BOOL : BOOL2BOOL(IN := true);
      SHOULD_NOT_FAIL : TEST_CONDITION;
    END_FBS
    EVENT_CONNECTIONS
      BOOL2BOOL.CNF TO SHOULD_NOT_FAIL.REQ;
      SHOULD_NOT_FAIL.CNF TO STEST_END.REQ;
    END_CONNECTIONS
    DATA_CONNECTIONS
      BOOL2BOOL.OUT TO SHOULD_NOT_FAIL.check;
    END_CONNECTIONS
  END_APPLICATION
  APPLICATION DeInitCommFB
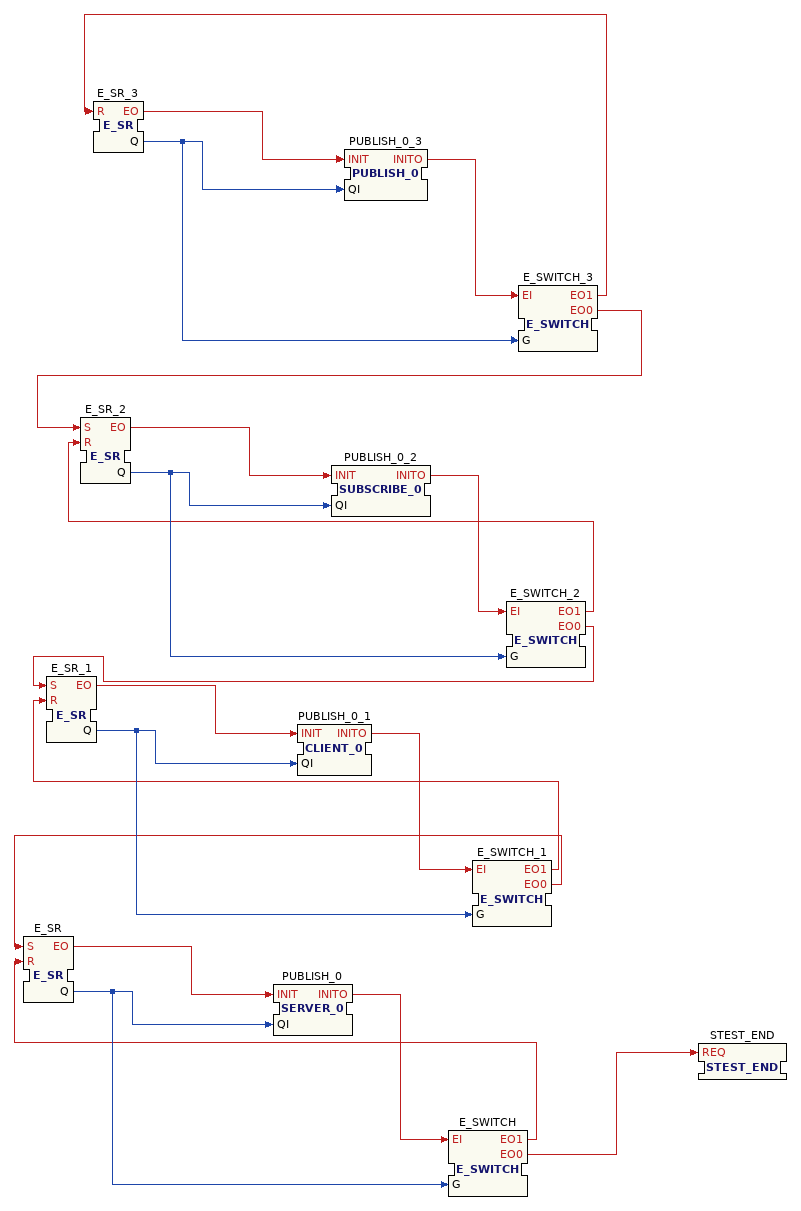
    FBS
      E_SR : E_SR;
      E_SWITCH : E_SWITCH;
      STEST_END : STEST_END;
      PUBLISH_0 : SERVER_0;
      E_SWITCH_1 : E_SWITCH;
      E_SR_1 : E_SR;
      E_SWITCH_2 : E_SWITCH;
      E_SR_2 : E_SR;
      E_SR_3 : E_SR;
      E_SWITCH_3 : E_SWITCH;
      PUBLISH_0_3 : PUBLISH_0;
      PUBLISH_0_2 : SUBSCRIBE_0;
      PUBLISH_0_1 : CLIENT_0;
    END_FBS
    EVENT_CONNECTIONS
      PUBLISH_0.INITO TO E_SWITCH.EI;
      E_SR_3.EO TO PUBLISH_0_3.INIT;
      PUBLISH_0_3.INITO TO E_SWITCH_3.EI;
      E_SR_2.EO TO PUBLISH_0_2.INIT;
      PUBLISH_0_2.INITO TO E_SWITCH_2.EI;
      E_SR_1.EO TO PUBLISH_0_1.INIT;
      PUBLISH_0_1.INITO TO E_SWITCH_1.EI;
      E_SWITCH_3.EO1 TO E_SR_3.R;
      E_SWITCH_3.EO0 TO E_SR_2.S;
      E_SWITCH_2.EO1 TO E_SR_2.R;
      E_SWITCH_2.EO0 TO E_SR_1.S;
      E_SWITCH_1.EO1 TO E_SR_1.R;
      E_SWITCH_1.EO0 TO E_SR.S;
      E_SWITCH.EO1 TO E_SR.R;
      E_SWITCH.EO0 TO STEST_END.REQ;
      E_SR.EO TO PUBLISH_0.INIT;
    END_CONNECTIONS
    DATA_CONNECTIONS
      E_SR.Q TO E_SWITCH.G;
      E_SR.Q TO PUBLISH_0.QI;
      E_SR_1.Q TO E_SWITCH_1.G;
      E_SR_2.Q TO E_SWITCH_2.G;
      E_SR_3.Q TO E_SWITCH_3.G;
      E_SR_3.Q TO PUBLISH_0_3.QI;
      E_SR_2.Q TO PUBLISH_0_2.QI;
      E_SR_1.Q TO PUBLISH_0_1.QI;
    END_CONNECTIONS
  END_APPLICATION
  APPLICATION simpleCommunicationTest
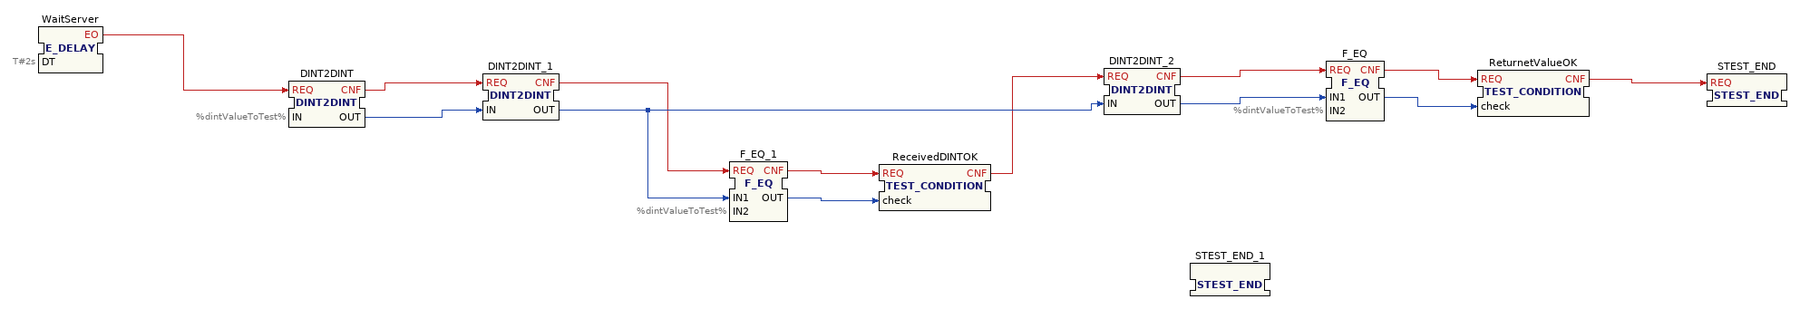
    FBS
      WaitServer : E_DELAY(DT := T#2s);
      ReturnetValueOK : TEST_CONDITION;
      F_EQ_1 : F_EQ(IN2 := %dintValueToTest%);
      F_EQ : F_EQ(IN2 := %dintValueToTest%);
      DINT2DINT_2 : DINT2DINT;
      DINT2DINT_1 : DINT2DINT;
      STEST_END : STEST_END;
      DINT2DINT : DINT2DINT(IN := %dintValueToTest%);
      ReceivedDINTOK : TEST_CONDITION;
      STEST_END_1 : STEST_END;
    END_FBS
    EVENT_CONNECTIONS
      DINT2DINT_1.CNF TO F_EQ_1.REQ;
      DINT2DINT.CNF TO DINT2DINT_1.REQ;
      ReceivedDINTOK.CNF TO DINT2DINT_2.REQ;
      F_EQ_1.CNF TO ReceivedDINTOK.REQ;
      F_EQ.CNF TO ReturnetValueOK.REQ;
      ReturnetValueOK.CNF TO STEST_END.REQ;
      DINT2DINT_2.CNF TO F_EQ.REQ;
      WaitServer.EO TO DINT2DINT.REQ;
    END_CONNECTIONS
    DATA_CONNECTIONS
      F_EQ_1.OUT TO ReceivedDINTOK.check;
      DINT2DINT_1.OUT TO DINT2DINT_2.IN;
      DINT2DINT.OUT TO DINT2DINT_1.IN;
      F_EQ.OUT TO ReturnetValueOK.check;
      DINT2DINT_1.OUT TO F_EQ_1.IN1;
      DINT2DINT_2.OUT TO F_EQ.IN1;
    END_CONNECTIONS
  END_APPLICATION
  APPLICATION CSVWriterTests
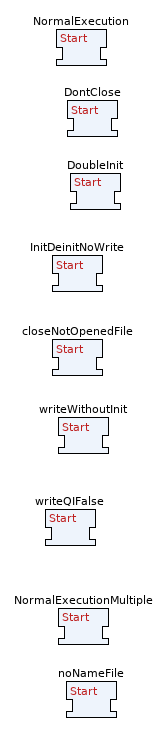
    SUBAPPLICATION NormalExecution
      EVENT_INPUT
        Start;
      END_EVENT
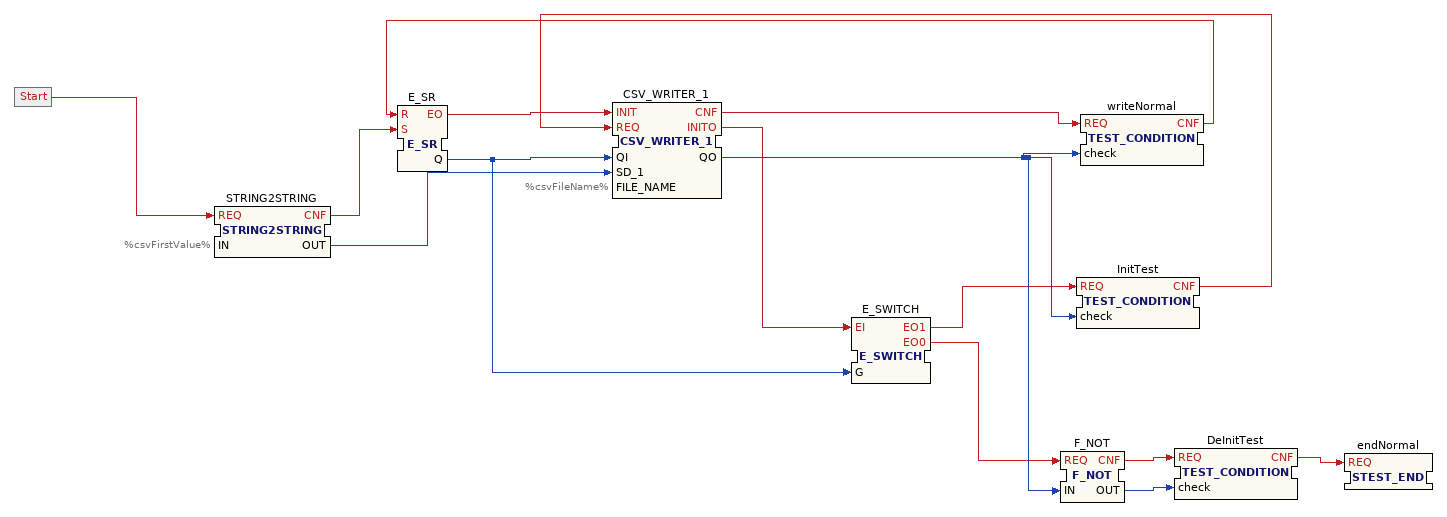
      FBS
        writeNormal : TEST_CONDITION;
        CSV_WRITER_1 : CSV_WRITER_1(FILE_NAME := %csvFileName%);
        InitTest : TEST_CONDITION;
        STRING2STRING : STRING2STRING(IN := %csvFirstValue%);
        DeInitTest : TEST_CONDITION;
        endNormal : STEST_END;
        F_NOT : F_NOT;
        E_SWITCH : E_SWITCH;
        E_SR : E_SR;
      END_FBS
      EVENT_CONNECTIONS
        CSV_WRITER_1.CNF TO writeNormal.REQ;
        writeNormal.CNF TO E_SR.R;
        E_SR.EO TO CSV_WRITER_1.INIT;
        InitTest.CNF TO CSV_WRITER_1.REQ;
        CSV_WRITER_1.INITO TO E_SWITCH.EI;
        E_SWITCH.EO1 TO InitTest.REQ;
        STRING2STRING.CNF TO E_SR.S;
        F_NOT.CNF TO DeInitTest.REQ;
        DeInitTest.CNF TO endNormal.REQ;
        E_SWITCH.EO0 TO F_NOT.REQ;
        Start TO STRING2STRING.REQ;
      END_CONNECTIONS
      DATA_CONNECTIONS
        CSV_WRITER_1.QO TO writeNormal.check;
        E_SR.Q TO CSV_WRITER_1.QI;
        STRING2STRING.OUT TO CSV_WRITER_1.SD_1;
        CSV_WRITER_1.QO TO InitTest.check;
        CSV_WRITER_1.QO TO F_NOT.IN;
        F_NOT.OUT TO DeInitTest.check;
        E_SR.Q TO E_SWITCH.G;
      END_CONNECTIONS
    END_SUBAPPLICATION
    SUBAPPLICATION DontClose
      EVENT_INPUT
        Start;
      END_EVENT
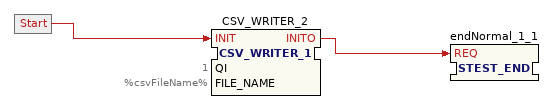
      FBS
        CSV_WRITER_2 : CSV_WRITER_1(QI := 1, FILE_NAME := %csvFileName%);
        endNormal_1_1 : STEST_END;
      END_FBS
      EVENT_CONNECTIONS
        CSV_WRITER_2.INITO TO endNormal_1_1.REQ;
        Start TO CSV_WRITER_2.INIT;
      END_CONNECTIONS
    END_SUBAPPLICATION
    SUBAPPLICATION DoubleInit
      EVENT_INPUT
        Start;
      END_EVENT
